TYPE "TAx_Warnings"
VERSION : 0.1
// Block: TAx_Warnings
   STRUCT
      TOAxis : Bool;
      Drive : Bool;
   END_STRUCT;

END_TYPE
